FUNCTION F_RawTimeToDCTimestruct : DCTimestruct
VAR_INPUT
	nRaw: ULINT;
	nUtcTimeBias: INT;
END_VAR
VAR
	fbTime: FB_ALY_DateTime;
END_VAR

fbTime.nRaw:= nRaw;
fbTime.nUtcTimeBias:= nUtcTimeBias;
F_RawTimeToDCTimestruct:= fbTime.stStructured;

END_FUNCTION

(* stored: POU F_RawTimeToDCTimestruct: Id 6ae3fafe-94b1-46ef-b50a-df71755a6923, SpecialFunc None *)
